Yaskawa INFORM job: FRONT_WELD_0ST-2_4940_V2.JBI

/JOB
//NAME FRONT_WELD_0ST-2_4940_V2
///FOLDERNAME 02-SKRZYNIE_JOBS
//POS
///NPOS 121,121,0,25,0,0
///TOOL 0
///POSTYPE PULSE
///PULSE
C00000=1212,-39190,49707,1936,-15809,-581
C00001=-55064,-17017,13106,20113,45767,-35735
C00002=-85641,-3161,12660,31281,67420,-55579
C00003=-77611,9747,38455,32702,57795,-55547
C00004=-77611,9747,38455,32702,57795,-55547
C00005=-80481,23547,61641,37204,60115,-56891
C00006=-80479,11681,28780,33754,71138,-52780
C00007=-72933,30277,53605,31576,73074,-55586
C00008=-73419,29451,52323,31530,73467,-55649
C00009=-73173,32098,57907,31817,71820,-56064
C00010=-72991,37471,72685,33001,66631,-57677
C00011=-82806,26311,53816,38180,73291,-53604
C00012=-71695,3747,16001,30713,64750,-51022
C00013=-70421,5575,20105,30867,63066,-51036
C00014=-35893,-19818,-4542,23004,50197,-40345
C00015=-37830,-23193,-8618,23571,50957,-40982
C00016=11136,-28839,-12562,1025,41780,-20887
C00017=20436,-26886,-6789,-12590,38175,-10721
C00018=58488,-10629,5191,-26833,51354,2977
C00019=55110,-17412,-5825,-19778,50988,-2825
C00020=79390,11759,28162,-35512,71262,52960
C00021=82927,23281,58968,-48274,65531,63493
C00022=83399,22743,58163,-48180,65853,63532
C00023=83221,24593,61395,-48465,65231,63817
C00024=82927,34411,85507,-52086,59386,67513
C00025=76815,18630,46530,-37158,64288,54543
C00026=79390,11759,28162,-35512,71262,52960
C00027=10831,-54278,-29128,-6468,39852,-5090
C00028=-67200,-10549,24402,-3189,24913,-39001
C00029=-75122,-2194,12822,3152,39225,-43427
C00030=-77516,10189,32861,8493,33365,-45533
C00031=-75154,17675,49539,7913,27349,-44943
C00032=-68113,10120,39417,1165,28259,-40458
C00033=-67114,5383,31515,9208,32648,-43213
C00034=-66450,3998,29285,10896,33890,-43630
C00035=-66374,3101,28136,14657,35566,-44954
C00036=-66747,-26,23691,26916,43760,-49061
C00037=-70537,4638,30761,35492,50867,-52773
C00038=-77050,-3138,8526,33226,61087,-51698
C00039=-67200,-10549,24402,-3189,24913,-39001
C00040=0,-52280,40443,83103,28146,-16510
C00041=99993,-20782,22705,-13349,24734,56519
C00042=67200,-10549,24402,3189,24913,39001
C00043=75122,-2194,12822,-3152,39225,43427
C00044=74323,5203,27259,-5972,33194,43789
C00045=74015,16414,48063,-6821,27325,44224
C00046=56519,1138,28747,9235,29393,33453
C00047=55467,619,28251,10155,29461,32830
C00048=56374,-724,25854,4078,30541,35419
C00049=56321,-6570,17381,-17816,37906,43384
C00050=68252,956,25699,-34035,49810,51639
C00051=77050,-3138,8526,-33226,61087,51698
C00052=67200,-10549,24402,3189,24913,39001
C00053=0,-52280,40443,-83103,28146,16510
C00054=-99993,-20782,22705,13349,24734,-56519
C00055=-91125,453,39555,30378,52425,-51131
C00056=-81425,-5449,14825,37552,56592,-47667
C00057=-81425,-10835,-2515,34915,62871,-45127
C00058=-79239,4305,16082,37593,68846,-50182
C00059=-83523,16585,41906,47112,68321,-58375
C00060=-83466,26209,67230,50527,61769,-62335
C00061=-83442,29914,76031,51903,59779,-63702
C00062=-84288,15645,43522,43516,65950,-57098
C00063=-90096,4679,14083,37467,76581,-51973
C00064=-87885,29238,52923,40761,81198,69685
C00065=-84355,23847,39024,40698,83720,72224
C00066=-82166,27958,47897,41071,80495,71788
C00067=-78317,33303,56220,41538,77506,72130
C00068=-90480,18737,31939,47254,81986,71631
C00069=-94217,10634,17426,46901,86469,-59967
C00070=-81425,-10835,-2515,34915,62871,-45127
C00071=-81425,-5449,14825,37552,56592,-47667
C00072=-94290,-610,44819,32366,49686,-53459
C00073=0,-55136,17047,60468,32096,-4233
C00074=99993,-20782,22705,-13349,24734,56519
C00075=91125,453,39555,-30378,52425,51131
C00076=81425,-5449,14825,-37552,56592,47667
C00077=81425,-10835,-2515,-34915,62871,45127
C00078=79239,4305,16082,-37593,68846,50182
C00079=80765,23031,47100,-43000,73595,58456
C00080=80765,35859,79857,-46269,64609,63023
C00081=81236,37975,84040,-46627,63953,63603
C00082=79256,17348,34699,-33448,76412,88212
C00083=79932,23608,50901,-39863,71219,88955
C00084=76220,30771,63034,-41386,67395,88927
C00085=86322,16060,37848,-39554,76452,89287
C00086=87424,-1569,9538,-38190,72401,52253
C00087=81425,-10835,-2515,-34915,62871,45127
C00088=92850,-11266,9233,-39092,60986,50964
C00089=28366,-40369,19479,-5635,23506,17663
C00090=-80334,-19501,31260,21216,42469,-40219
C00091=-80621,-32280,-9061,25825,59412,-41877
C00092=-80621,-37319,-22868,24573,64555,-40576
C00093=-75108,-2453,16462,35304,60348,-42510
C00094=-72509,6961,33136,36537,55809,-43202
C00095=-35516,-19804,6201,28214,41034,-31537
C00096=-39606,-22901,-1163,28356,44724,-32188
C00097=15344,-29112,-5358,-2858,33820,-6852
C00098=13899,-24312,2834,-1929,31756,-7563
C00099=57847,-8649,16006,-27199,42364,12903
C00100=60973,-17187,4937,-27817,44388,13718
C00101=60973,-17187,4937,-27817,44388,13718
C00102=-13287,-42463,-12044,19170,31021,-23010
C00103=-32327,-13779,23475,31826,45619,-34841
C00104=-7543,-16914,18595,22802,40898,-24102
C00105=-14713,-8676,25653,29650,51413,-29764
C00106=10328,-9633,21800,22575,44712,-20445
C00107=17643,-12152,18299,16053,41434,-15515
C00108=30651,-6482,23782,13822,41017,-11573
C00109=64054,-19541,3059,-29141,44956,15011
C00110=51466,-33957,-1499,-46586,51805,23434
C00111=51968,11221,64546,-46494,62445,32842
C00112=17724,-9538,26927,-32521,50696,25771
C00113=30460,-1291,51024,-52582,52656,27640
C00114=3648,-6440,45181,-59097,38550,24318
C00115=-779,-7616,40691,-53947,37163,20579
C00116=-19026,-3257,48764,-59965,27841,19640
C00117=-71680,-19835,10874,33863,39440,-36917
C00118=-20806,-37586,-12792,9951,42782,-18031
///LIMIT ON
C00119=29087,-45372,27330,-13325,19529,9021
C00120=0,-35121,73515,0,-2982,0
///LIMIT OFF
BC00000=817112
BC00001=869064
BC00002=872323
BC00003=872323
BC00004=872323
BC00005=872323
BC00006=889185
BC00007=889187
BC00008=889187
BC00009=889187
BC00010=889187
BC00011=889187
BC00012=889187
BC00013=889187
BC00014=889187
BC00015=889187
BC00016=889187
BC00017=889186
BC00018=889187
BC00019=889188
BC00020=889188
BC00021=889186
BC00022=889186
BC00023=889186
BC00024=889186
BC00025=889188
BC00026=889188
BC00027=884698
BC00028=860846
BC00029=890023
BC00030=890026
BC00031=890026
BC00032=890023
BC00033=890024
BC00034=890025
BC00035=890025
BC00036=890026
BC00037=890026
BC00038=890026
BC00039=860846
BC00040=789452
BC00041=789452
BC00042=860846
BC00043=890023
BC00044=890026
BC00045=890026
BC00046=890026
BC00047=890026
BC00048=890031
BC00049=890038
BC00050=890027
BC00051=890026
BC00052=860846
BC00053=789452
BC00054=789452
BC00055=826914
BC00056=872717
BC00057=892114
BC00058=892116
BC00059=892116
BC00060=892116
BC00061=892116
BC00062=892116
BC00063=892692
BC00064=892116
BC00065=906055
BC00066=906055
BC00067=906055
BC00068=906055
BC00069=906055
BC00070=892114
BC00071=872717
BC00072=826914
BC00073=827200
BC00074=789452
BC00075=826914
BC00076=872717
BC00077=892114
BC00078=892116
BC00079=892116
BC00080=892116
BC00081=892116
BC00082=892116
BC00083=892116
BC00084=892116
BC00085=892116
BC00086=892116
BC00087=892114
BC00088=872717
BC00089=803729
BC00090=818207
BC00091=837767
BC00092=876072
BC00093=876072
BC00094=876072
BC00095=876070
BC00096=876072
BC00097=876072
BC00098=876072
BC00099=876070
BC00100=876072
BC00101=868737
BC00102=876072
BC00103=876072
BC00104=876068
BC00105=876068
BC00106=876070
BC00107=876114
BC00108=876070
BC00109=876072
BC00110=876072
BC00111=876068
BC00112=876070
BC00113=876073
BC00114=876073
BC00115=876072
BC00116=876072
BC00117=876072
BC00118=872664
BC00119=759440
BC00120=651598
///POSTYPE BASE
///RECTAN
///RCONF 0,0,0,0,0,0,0,0,0,0,0,0,0,0,0,0,0,0,0,0,0,0,0,0
P00021=6.550,-0.003,-5.735,0.0000,0.0000,0.0000
P00022=5.943,-0.018,-6.388,0.0000,0.0000,0.0000
P00023=7.025,-0.019,-7.168,0.0000,0.0000,0.0000
P00024=5.926,-0.047,-4.777,0.0000,0.0000,0.0000
P00350=11.519,-0.008,1.149,0.0000,0.0000,0.0000
P00351=13.563,-0.027,-0.653,0.0000,0.0000,0.0000
P00352=13.252,-0.027,-0.827,0.0000,0.0000,0.0000
P00353=10.971,-0.082,0.776,0.0000,0.0000,0.0000
P00399=-2.449,0.031,8.825,0.0000,0.0000,0.0000
P00400=5.920,-3.503,-0.024,0.0000,0.0000,0.0000
P00401=3.430,-0.021,1.131,0.0000,0.0000,0.0000
P00402=-0.253,1.107,3.062,0.0000,0.0000,0.0000
P00403=-3.666,-0.015,5.328,0.0000,0.0000,0.0000
P00405=2.420,0.007,1.427,0.0000,0.0000,0.0000
P00406=3.513,-0.022,0.429,0.0000,0.0000,0.0000
P00415=-1.781,-1.303,3.250,0.0000,0.0000,0.0000
P00416=0.027,1.119,3.078,0.0000,0.0000,0.0000
P00420=-0.017,0.555,2.209,0.0000,0.0000,0.0000
P00421=4.378,0.044,2.315,0.0000,0.0000,0.0000
P00422=2.474,0.026,-1.450,0.0000,0.0000,0.0000
P00423=4.044,0.004,-2.619,0.0000,0.0000,0.0000
P00424=-0.387,-0.003,1.304,0.0000,0.0000,0.0000
P00425=-1.050,0.029,1.708,0.0000,0.0000,0.0000
P00426=0.002,-0.749,-0.024,0.0000,0.0000,0.0000
P00427=-1.030,-0.025,3.232,0.0000,0.0000,0.0000
//INST
///DATE 2025/04/15 14:44
///ATTR SC,RW
///GROUP1 RB1,BS1
NOP
'**********************
'**********************
'POCZATEK SPAWANIA PRZOD
'**********************
'**********************
MOVJ C00000 BC00000 VJ=60.00
MOVL C00001 BC00001 V=416.7
MOVJ C00002 BC00002 VJ=10.00
MOVJ C00003 BC00003 VJ=10.00
MOVL C00004 BC00004 V=150.0
MOVL C00005 BC00005 V=150.0
'**********************
'W41A SIDE
'**********************
MOVL C00006 BC00006 V=250.0
SFTON P0402
MOVL C00007 BC00007 V=66.7 PL=0
REFP 1 C00008 BC00008
REFP 2 C00009 BC00009
MACRO1 MJ#(0) ARGF14
ARCON
WVON WEV#(5)
MOVL C00010 BC00010 V=9.2
ARCOF
WVOF
SFTOF
MOVL C00011 BC00011 V=166.7
'**********************
'W41A FRONT
'**********************
MOVL C00012 BC00012 V=250.0
SFTON P0350
MOVL C00013 BC00013 V=66.7 PL=0
SFTOF
MACRO1 MJ#(0) ARGF21
ARCON
WVON WEV#(2)
SFTON P0351
MOVL C00014 BC00014 V=8.3
SFTOF
ARCOF
WVOF
MOVL C00015 BC00015 V=166.7
'**********************
'W41B FRONT
'**********************
MOVL C00016 BC00016 V=250.0
SFTON P0352
MOVL C00017 BC00017 V=66.7 PL=0
SFTOF
MACRO1 MJ#(0) ARGF21
ARCON
WVON WEV#(2)
SFTON P0353
MOVL C00018 BC00018 V=8.3
SFTOF
ARCOF
WVOF
MOVL C00019 BC00019 V=166.7
MOVL C00020 BC00020 V=100.0
'**********************
'W41A SIDE
'**********************
SFTON P0400
MOVL C00021 BC00021 V=66.7 PL=0
MACRO1 MJ#(0) ARGF21
REFP 1 C00022 BC00022
REFP 2 C00023 BC00023
ARCON
WVON WEV#(5)
MOVL C00024 BC00024 V=8.3
ARCOF
WVOF
SFTOF
MOVL C00025 BC00025 V=166.7
MOVL C00026 BC00026 V=166.7
MOVL C00027 BC00027 V=333.3
MOVJ C00028 BC00028 VJ=20.00
MOVJ C00029 BC00029 VJ=20.00
'**********************
'W42A.1
'**********************
'POPRAWIC
MOVL C00030 BC00030 V=500.0
SFTON P0403
MOVL C00031 BC00031 V=66.7 PL=0
MACRO1 MJ#(0) ARGF9
ARCON
MOVL C00032 BC00032 V=9.2
SFTON P0416
MOVL C00033 BC00033 V=9.2
MOVL C00034 BC00034 V=9.2
MOVL C00035 BC00035 V=9.2
SFTON P0421
MOVL C00036 BC00036 V=9.2
SFTON P0402
MOVL C00037 BC00037 V=9.2
ARCOF
MOVL C00038 BC00038 V=500.0
SFTOF
MOVJ C00039 BC00039 VJ=15.00
'W42B.1
MOVJ C00040 BC00040 VJ=30.00
MOVJ C00041 BC00041 VJ=30.00
MOVJ C00042 BC00042 VJ=30.00
MOVJ C00043 BC00043 VJ=30.00
'**********************
'W42B.1
'**********************
MOVL C00044 BC00044 V=500.0
SFTON P0399
MOVL C00045 BC00045 V=166.7 PL=0
MACRO1 MJ#(0) ARGF9
ARCON
SFTON P0415
MOVL C00046 BC00046 V=9.2
MOVL C00047 BC00047 V=9.2
MOVL C00048 BC00048 V=9.2
SFTON P0427
MOVL C00049 BC00049 V=9.2
SFTON P0400
MOVL C00050 BC00050 V=9.2
ARCOF
MOVL C00051 BC00051 V=500.0
SFTOF
MOVJ C00052 BC00052 VJ=25.00
'W42A.2
MOVJ C00053 BC00053 VJ=40.00
MOVJ C00054 BC00054 VJ=30.00
MOVJ C00055 BC00055 VJ=30.00
MOVJ C00056 BC00056 VJ=30.00
MOVJ C00057 BC00057 VJ=30.00
'**********************
'W42A.2
'**********************
MOVL C00058 BC00058 V=500.0
SFTON P0420
MOVL C00059 BC00059 V=166.7 PL=0
SFTOF
MACRO1 MJ#(0) ARGF9
ARCON
WVON WEV#(6)
MOVL C00060 BC00060 V=9.2
SFTON P0402
MOVL C00061 BC00061 V=9.2
ARCOF
WVOF
MOVL C00062 BC00062 V=166.7
MOVJ C00063 BC00063 VJ=20.00
MOVJ C00064 BC00064 VJ=20.00
MOVL C00065 BC00065 V=250.0
MOVL C00066 BC00066 V=166.7
ARCON
MOVL C00067 BC00067 V=10.8
ARCOF
MOVL C00068 BC00068 V=166.7
MOVJ C00069 BC00069 VJ=20.00
SFTOF
MOVJ C00070 BC00070 VJ=30.00
MOVJ C00071 BC00071 VJ=30.00
MOVJ C00072 BC00072 VJ=30.00
'W42B.2
MOVJ C00073 BC00073 VJ=30.00
MOVJ C00074 BC00074 VJ=30.00
MOVJ C00075 BC00075 VJ=30.00
MOVJ C00076 BC00076 VJ=30.00
MOVJ C00077 BC00077 VJ=30.00
'**********************
'W42B.2
'**********************
MOVL C00078 BC00078 V=500.0
SFTON P0426
MOVL C00079 BC00079 V=166.7 PL=0
SFTOF
MACRO1 MJ#(0) ARGF9
ARCON
WVON WEV#(6)
MOVL C00080 BC00080 V=9.2
SFTON P0400
MOVL C00081 BC00081 V=9.2
ARCOF
WVOF
SFTOF
MOVJ C00082 BC00082 VJ=10.00
SFTON P0400
MOVL C00083 BC00083 V=166.7
ARCON
MOVL C00084 BC00084 V=10.8
ARCOF
MOVL C00085 BC00085 V=250.0
MOVL C00086 BC00086 V=500.0
SFTOF
MOVJ C00087 BC00087 VJ=20.00
MOVJ C00088 BC00088 VJ=30.00
'W42A.3
MOVJ C00089 BC00089 VJ=20.00
MOVJ C00090 BC00090 VJ=20.00
MOVJ C00091 BC00091 VJ=30.00
MOVJ C00092 BC00092 VJ=30.00
'**********************
'W42A.3
'**********************
MOVL C00093 BC00093 V=500.0
SFTON P0021
MOVL C00094 BC00094 V=166.7 PL=0
MACRO1 MJ#(0) ARGF9
ARCON
WVON WEV#(2)
SFTON P0022
MOVL C00095 BC00095 V=9.2
ARCOF
WVOF
MOVL C00096 BC00096 V=500.0
SFTOF
'**********************
'W42B.3
'**********************
MOVL C00097 BC00097 V=500.0
SFTON P0023
MOVL C00098 BC00098 V=166.7 PL=0
ARCON
WVON WEV#(2)
SFTON P0024
MOVL C00099 BC00099 V=9.2
ARCOF
WVOF
MOVL C00100 BC00100 V=500.0
SFTOF
MOVJ C00101 BC00101 VJ=20.00
'**********************
'GORA L
'**********************
MOVL C00102 BC00102 V=500.0
SFTON P0401
MOVL C00103 BC00103 V=166.7 PL=0
MACRO1 MJ#(0) ARGF9
ARCON
MOVL C00104 BC00104 V=11.7
SFTON P0424
MOVL C00105 BC00105 V=11.7
SFTON P0425
MOVL C00106 BC00106 V=11.7
SFTON P0406
MOVL C00107 BC00107 V=11.7
MOVL C00108 BC00108 V=11.7
ARCOF
MOVL C00109 BC00109 V=500.0
SFTOF
'**********************
'GORA P
'**********************
MOVL C00110 BC00110 V=166.7
SFTON P0401
MOVL C00111 BC00111 V=166.7 PL=0
ARCON
MOVL C00112 BC00112 V=11.7
SFTON P0423
MOVL C00113 BC00113 V=11.7
SFTON P0422
MOVL C00114 BC00114 V=11.7
SFTON P0405
MOVL C00115 BC00115 V=11.7
MOVL C00116 BC00116 V=11.7
ARCOF
MOVL C00117 BC00117 V=500.0
SFTOF
MOVJ C00118 BC00118 VJ=20.00
MOVJ C00119 BC00119 VJ=30.00
MOVJ C00120 BC00120 VJ=30.00
'KONIEC SPAWANIA FRONTU
END
